# EPICS autosave request: iocBoot/iocdelaygen/autosave/auto_settings.req
## DG645 digital delay generator settings
file drvDG645_settings.req P=$(P),R=DG0:
